FUNCTION FC_ProductStatusDatabase : eDbPiecesStatus
VAR_INPUT
	In					: STRING(50);
END_VAR

IF In = 'Completed' THEN
	FC_ProductStatusDatabase := eDbPiecesStatus.Completed;
ELSIF In = 'Scrap' THEN
	FC_ProductStatusDatabase := eDbPiecesStatus.Scrap;
ELSIF In = 'Processing' THEN
	FC_ProductStatusDatabase := eDbPiecesStatus.Processing;
ELSIF In = 'Fetched' THEN
	FC_ProductStatusDatabase := eDbPiecesStatus.Fetched;
ELSIF In = 'Undefined' THEN
	FC_ProductStatusDatabase := eDbPiecesStatus.Undefined;
ELSE
	FC_ProductStatusDatabase := eDbPiecesStatus.Undefined;
END_IF

END_FUNCTION

(* stored: Version 1.1.0.1, ProductVersion 3.1.4024.15
   POU FC_ProductStatusDatabase: Id {94f9f019-117f-4481-8e82-88a9977c1fa4}, SpecialFunc None *)
